FUNCTION_BLOCK FB_AxisConfig
VAR_INPUT
	bExecute: BOOL; // Set, then get
	bExecGet: BOOL; // Only get
	bReset: BOOL;
	stConfigSet: ST_AxisParams;
	stHardware: ST_AxisHardware;
END_VAR
VAR_IN_OUT
	Axis: AXIS_REF;
END_VAR
VAR_OUTPUT
	bDone: BOOL;
	bValid: BOOL;
	bBusy: BOOL;
	bError: BOOL;
	nErrorID: UDINT;
	bInitDone: BOOL;
	bInitPreOp: BOOL;
	stConfigGet: ST_AxisParams;
END_VAR
VAR
	fbRead: FB_AxisReadParams;
	fbWrite: FB_AxisWriteParams;
	bDoRead: BOOL;
END_VAR

// Write first
fbWrite(bExecute:=bExecute,
	bReset:=bReset,
	stConfig:=stConfigSet,
	stHardware:=stHardware,
	Axis:=Axis);
// Can only be turned on! Not back off!
IF fbWrite.bInitPreOp THEN
	bInitPreOP := TRUE;
END_IF
// Reset bDoRead if both execs are false
IF NOT bExecute AND NOT bExecGet THEN
	bDoRead := FALSE;
END_IF
// If bExecute is TRUE, wait untill after the write to read
IF bExecute THEN
	bDoRead := fbWrite.bDone;
ELSE
	bDoRead := bExecGet;
END_IF
// Notify that its ok to set master to OP.
// This block is really only used if we skip the write step.
IF bDoRead THEN
	bInitPreOP := TRUE;
END_IF
// Read now
fbRead(bExecute:=bDoRead,
	bReset:=bReset,
	stHardware:=stHardware,
	Axis:=Axis,
	stConfig=>stConfigGet,
	bValid=>bValid);
// Set the status outputs
IF bExecute THEN
	bDone := fbWrite.bDone AND NOT fbRead.bBusy;
ELSIF bExecGet THEN
	bDone := NOT fbRead.bBusy;
ELSE
	bDone := FALSE;
END_IF
bBusy := fbWrite.bBusy OR fbRead.bBusy;
bError := fbWrite.bError OR fbRead.bError;
IF fbWrite.nErrorID > 0 THEN
	nErrorID := fbWrite.nErrorID;
ELSE
	nErrorID := fbRead.nErrorID;
END_IF
IF bDone THEN
	bInitDone := TRUE;
END_IF
IF bError THEN
	bInitDone := FALSE;
END_IF
IF bReset THEN
	bReset := FALSE;
END_IF

END_FUNCTION_BLOCK

(* stored: Version 1.1.0.1, ProductVersion 3.1.4020.14
   POU FB_AxisConfig: Id {fcb6a2ad-e399-41e9-a4d8-8a9b39418313}, SpecialFunc None *)
